FUNCTION_BLOCK FB_PowerModeConditioningSFC
VAR_IN_OUT
	//IPSState						:	ST_InternalPowerStatus;
	IPSDemand						:	ST_PowerDemand;
	
	ConditioningRequirements		: 	ST_ConditioningRequirements;
	Control							:	ST_CoolingSystem_Control;
	Get								:	ST_CoolingSystemGet;	

END_VAR
VAR_OUTPUT
	SFCActive	:	BOOL;
END_VAR

VAR
	AverageSystemLoadData	:	ARRAY[0..240] OF LREAL;
	// Gemiddelde load over 60s, Koelsysteem is toch traag
	AverageSystemLoadParams : TC2_ControllerToolbox.ST_CTRL_MOVING_AVERAGE_PARAMS := (tCtrlCycleTime := TIME#250ms, tTaskCycleTime := TIME#250ms, nSamplesToFilter := 240, pWorkArray_ADR := ADR(AverageSystemLoadData), nWorkArray_SIZEOF := sizeof(AverageSystemLoadData));
	AverageSystemLoad: FB_CTRL_MOVING_AVERAGE;
	
	CorrectionPIDParams : TC2_ControllerToolbox.ST_CTRL_PID_PARAMS := (tCtrlCycleTime := CoolingSystemParams.PIDLoopTime, tTaskCycleTime := CoolingSystemParams.PIDLoopTime, fKp := CoolingSystemParams.PIDControlKfactor, tTn := CoolingSystemParams.PIDControlTn, tTv := CoolingSystemParams.PIDControlTv, tTd := CoolingSystemParams.PIDControlTd, fOutMaxLimit := CoolingSystemParams.PIDControlLimitMax, fOutMinLimit := CoolingSystemParams.PIDControlLimitMin);
	CorrectionPID: FB_CTRL_PID;
	//NewSetpoint: REAL;
	
	r_ExpectedBaseCoolantTemp	:	REAL;
	
	b_ValveStateOK	:	Bool;
END_VAR

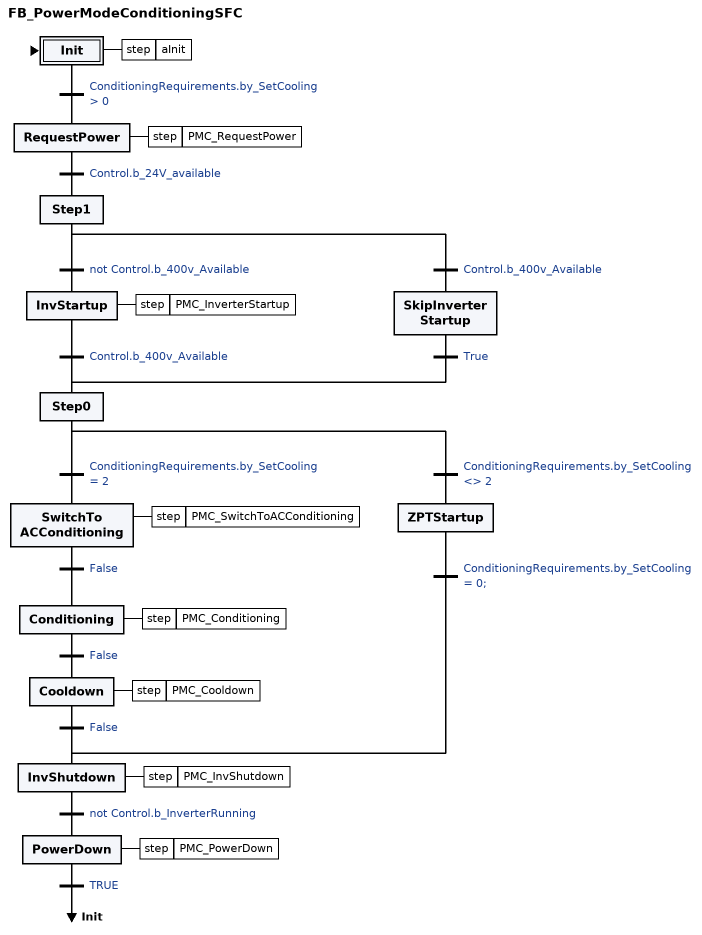
INITIAL_STEP Init:
    aInit(N);  // step action
END_STEP
TRANSITION FROM Init TO RequestPower
    := ConditioningRequirements.by_SetCooling > 0;
END_TRANSITION
STEP RequestPower:
    PMC_RequestPower(N);  // step action
END_STEP
TRANSITION FROM RequestPower TO Step1
    := Control.b_24V_available;
END_TRANSITION
STEP Step1:
END_STEP
TRANSITION FROM Step1 TO InvStartup
    := not Control.b_400v_Available;
END_TRANSITION
STEP InvStartup:
    PMC_InverterStartup(N);  // step action
END_STEP
TRANSITION FROM InvStartup TO Step0
    := Control.b_400v_Available;
END_TRANSITION
TRANSITION FROM Step1 TO SkipInverterStartup
    := Control.b_400v_Available;
END_TRANSITION
STEP SkipInverterStartup:
END_STEP
TRANSITION FROM SkipInverterStartup TO Step0
    := True;
END_TRANSITION
STEP Step0:
END_STEP
TRANSITION FROM Step0 TO SwitchToACConditioning
    := ConditioningRequirements.by_SetCooling = 2;
END_TRANSITION
STEP SwitchToACConditioning:
    PMC_SwitchToACConditioning(N);  // step action
END_STEP
TRANSITION FROM SwitchToACConditioning TO Conditioning
    := False;
END_TRANSITION
STEP Conditioning:
    PMC_Conditioning(N);  // step action
END_STEP
TRANSITION FROM Conditioning TO Cooldown
    := False;
END_TRANSITION
STEP Cooldown:
    PMC_Cooldown(N);  // step action
END_STEP
TRANSITION FROM Cooldown TO InvShutdown
    := False;
END_TRANSITION
TRANSITION FROM Step0 TO ZPTStartup
    := ConditioningRequirements.by_SetCooling <> 2;
END_TRANSITION
STEP ZPTStartup:
END_STEP
TRANSITION FROM ZPTStartup TO InvShutdown
    := ConditioningRequirements.by_SetCooling = 0;
END_TRANSITION
STEP InvShutdown:
    PMC_InvShutdown(N);  // step action
END_STEP
TRANSITION FROM InvShutdown TO PowerDown
    := not Control.b_InverterRunning;
END_TRANSITION
STEP PowerDown:
    PMC_PowerDown(N);  // step action
END_STEP
TRANSITION FROM PowerDown TO Init
    := TRUE;
END_TRANSITION
// branch label Branch0_PowerModeSFC

ACTION aInit:
SFCActive := False;
END_ACTION

ACTION PMC_Conditioning:


{warning "PowerModePID nog uitwerken en testen"}
{warning "placeholder voor de pid"}
// PID testen kan pas als het systeem helemaal draait. Voor nu geen tijd in stoppen maar testen met fixed setpoint.
//Gezien de modulerende regeling van de warmtepomp is een uitgebreide PID misschien amper nodig, enkel een long-term reactie op daadwerkelijke accutemperatuur.

Control.e_HeatpumpMode := eHeatpumpMode.Cooling;
Control.r_HeatPumpSetpoint := 10.0;

//initiate cooldown
IF ConditioningRequirements.by_SetCooling < 2 THEN
	ConditioningRequirements.by_PSCoolingPowerMode := 1;
	SFCTip := TRUE;
END_IF

//if coolantpressure drops below startup minimum, start DC pump and shutdown system immediately!
IF Control.r_CoolantPressure < (CoolingSystemParams.StartupPumpMinimumPressure + Control.r_CoolantIdlePressure) THEN
	control.b_DCPumpEnable := TRUE;
	get.Events.b_InverterCoolingLoopError := TRUE;
	ConditioningRequirements.by_PSCoolingPowerMode := 0;
END_IF


//PID disabled for now. Test with fixed setpoint first.


//AverageSystemLoad(stParams := AverageSystemLoadParams, fIn := Control.r_OutputPowerLevel);
//r_ExpectedBaseCoolantTemp := LREAL_TO_REAL(CoolingSystemParams.BattGoalTemp-(AverageSystemLoad.fOut /100 * CoolingSystemParams.CoolantFullPowerTemperatureOffset));

//Coolingsystem dictated by battery
//CorrectionPID.stParams := CorrectionPIDParams;
//CorrectionPID.fSetpointValue := CoolingSystemParams.BattGoalTemp;
//CorrectionPID.fActualValue := BattAvgTemp;

//CorrectionPID.stParams.fKp := CoolingSystemParams.PIDControlKfactor;

//CorrectionPID.stParams.tCtrlCycleTime := CoolingSystemParams.PIDLoopTime;
//CorrectionPID.stParams.tTn := CoolingSystemParams.PIDControlTn;//Integral coefficient
//CorrectionPID.stParams.tTv := CoolingSystemParams.PIDControlTv;//Derivative coefficient 
//CorrectionPID.stParams.tTd := CoolingSystemParams.PIDControlTd;//Damping time 
//CorrectionPID.stParams.fOutMaxLimit := CoolingSystemParams.PIDControlLimitMax;      //max correctie
//CorrectionPID.stParams.fOutMinLimit := CoolingSystemParams.PIDControlLimitMin;     // min correctie 
//CorrectionPID.stParams.bDInTheFeedbackPath := FALSE; //voorkomt oscillatie bij setpoint wijziging door dif loop. maar die is hier niet in gebruik.
//CorrectionPID.stParams.bPInTheFeedbackPath := FALSE; //?


//CorrectionPID(	stParams := CorrectionPIDParams, 
//				fSetpointValue := CoolingSystemParams.BattGoalTemp, 
//				fActualValue := Control.r_BMSBatteryTemperature);
				

//Control.r_HeatPumpSetpoint := r_ExpectedBaseCoolantTemp - CorrectionPID.fOut;
END_ACTION

ACTION PMC_Cooldown:

//first setup. Basic setpoint to return to idle temperatures
// After battery is done, enclosure is checked as well. May not be neccessary.
//Inverter is currently not checked, may be desirable after long runs.

IF ConditioningRequirements.Battery = eConditioningRequirement.Cooling THEN
	Control.b_CloseBatteryLoopValve := FALSE;
	Control.e_HeatpumpMode := eHeatpumpmode.Cooling;
	Control.r_HeatPumpSetpoint := 10.0;
ELSIF ConditioningRequirements.Battery = eConditioningRequirement.Heating THEN
	Control.b_CloseBatteryLoopValve := FALSE;
	Control.e_HeatpumpMode := eHeatpumpmode.Heating;
	Control.r_HeatPumpSetpoint := 35.0;
ELSE
	//battery conditioning done, close valve to speed up other conditioning loops
	Control.b_CloseBatteryLoopValve := TRUE;
	IF ConditioningRequirements.Enclosure = eConditioningRequirement.Heating THEN
		Control.e_HeatpumpMode := eHeatpumpmode.Heating;
		Control.r_HeatPumpSetpoint := 35.0;
	ELSIF ConditioningRequirements.Enclosure = eConditioningRequirement.Cooling THEN
		Control.e_HeatpumpMode := eHeatpumpmode.Cooling;
		Control.r_HeatPumpSetpoint := 10.0;
	ELSE
		//if enclosure and battery are ok. Inverter is presumably already cooled down enough. 
		Control.e_HeatpumpMode := eHeatpumpmode.standby;
		SFCTip := TRUE;	

	{warning "Add inverter temp check?"};
	//If not, keep running in current mode for longer
	//	IF PSGet.r_TemperatureMax < CoolingSystemParams.InverterIdleShutdownTemp THEN
		//	ConditioningModeRequired := eConditioningStates.OFF;
		//END_IF
	END_IF	
END_IF
END_ACTION

ACTION PMC_InverterStartup:
Control.b_CloseBatteryLoopValve 	:= TRUE;
Control.b_CloseFancoilLoopValve 	:= TRUE;
Control.b_CloseInverterLoopValve 	:= FALSE;

Control.b_DCFancoilEnable := FALSE;
//Control.b_ACFancoilEnable := FALSE;

Control.b_DCPumpEnable := TRUE;
Control.b_ACPumpEnable := FALSE;


Control.b_HeatPumpPowerEnable := FALSE;

//if both are ok, the inverter should have enough flow to start
IF Control.r_CoolantPressure > (CoolingSystemParams.StartupPumpMinimumPressure + Control.r_CoolantIdlePressure) AND Control.b_InverterLoopEnabled THEN
	//Inverter may commence modulating, but no power delivery yet.
	ConditioningRequirements.by_PSCoolingPowerMode := 1;
END_IF
END_ACTION

ACTION PMC_InvShutdown:
Control.b_CloseBatteryLoopValve := TRUE;
Control.b_CloseFancoilLoopValve := TRUE;
Control.b_CloseBatteryLoopValve := FALSE;

Control.b_DCFancoilEnable := FALSE;
//Control.b_ACFancoilEnable := FALSE;

Control.b_DCPumpEnable := TRUE;
Control.b_ACPumpEnable := FALSE;

Control.b_HeatPumpPowerEnable := FALSE;
Control.e_HeatpumpMode := eHeatpumpmode.standby;

//Inverter may shutdown now
ConditioningRequirements.by_PSCoolingPowerMode := 0;
END_ACTION

ACTION PMC_PowerDown:

Control.b_CloseBatteryLoopValve 	:= FALSE;
Control.b_CloseFancoilLoopValve 	:= FALSE;
Control.b_CloseBatteryLoopValve 	:= FALSE;

Control.b_DCFancoilEnable 		:= FALSE;
//Control.b_ACFancoilEnable		:= FALSE;

Control.b_DCPumpEnable 			:= FALSE;
Control.b_ACPumpEnable 			:= FALSE;

Control.b_HeatPumpPowerEnable	:= FALSE;


IPSDemand.b_Demand_24V 			:= FALSE;

SFCActive := FALSE;
END_ACTION

ACTION PMC_RequestPower:
SFCActive := TRUE;
IPSDemand.b_Demand_24V := TRUE;
IPSDemand.b_Demand_400V := TRUE;
END_ACTION

ACTION PMC_SwitchToACConditioning:





//First enable both pumps to see if AC pump works (by checking pressure increase)
Control.b_ACPumpEnable 			:= TRUE;
Control.b_DCPumpEnable 			:= TRUE;

IF Control.r_CoolantPressure > (CoolingSystemParams.MainPumpMinimumPressure + Control.r_CoolantIdlePressure) THEN
	Control.b_CloseBatteryLoopValve 	:= FALSE;
	Control.b_CloseFancoilLoopValve 	:= FALSE;
	Control.b_CloseInverterLoopValve 	:= FALSE;
		
	Control.b_HeatPumpPowerEnable 	:= TRUE;
	Control.e_HeatpumpMode := eHeatpumpmode.standby;
	
	Control.b_DCPumpEnable 			:= FALSE;
	
	Control.b_DCFancoilEnable 		:= TRUE;

	//if all loops are enabled, system is ready for operation
	IF Control.b_BatteryLoopEnabled AND Control.b_InverterLoopEnabled AND Control.b_FancoilLoopEnabled THEN;
		ConditioningRequirements.by_PSCoolingPowerMode := 2;
		SFCTip := TRUE;
	END_IF
END_IF
END_ACTION

METHOD SFCEnable : BOOL
VAR_INPUT
	Enable	:	Bool;
END_VAR
IF Enable THEN
	SFCInit := FALSE;
ELSE
	SFCActive:= FALSE;
	SFCInit := TRUE;
END_IF
END_METHOD

END_FUNCTION_BLOCK

(* stored: Version 1.1.0.1, ProductVersion 3.1.4024.12
   POU FB_PowerModeConditioningSFC: Id {3d14e69f-c7d5-448c-91d8-2523ca0c80a5}, SpecialFunc None
   Action aInit: Id {6929f8a4-59b4-47f7-be18-5afa05fbaf8d}
   Action PMC_Conditioning: Id {8bbaaefd-56bb-4f8a-ab3d-6150c32a933c}
   Action PMC_Cooldown: Id {df814817-b8e8-4a1c-b70a-ae3074173fbe}
   Action PMC_InverterStartup: Id {ec99f816-b172-4523-ba49-4230b1a52a65}
   Action PMC_InvShutdown: Id {b3bf1e48-af19-4633-90a1-52a71a2560a3}
   Action PMC_PowerDown: Id {0cef10fc-975e-4cea-97c1-bd5025fb310a}
   Action PMC_RequestPower: Id {8b6c7fd9-4f84-4ee2-bb44-cf6f066a947f}
   Action PMC_SwitchToACConditioning: Id {ae7c7307-7c32-44c0-9dcd-c663e74a0231}
   Method SFCEnable: Id {c670328c-4d51-4811-acc1-a4e98b706f4f} *)
